FUNCTION Filtro : REAL
VAR_INPUT
	Input:REAL;	//Entrada do sensor
	Tempo:DINT := 500;	//Tempo de amostragem
END_VAR
VAR
	Amostras:ARRAY[1..50] OF REAL;
	TON_Amostras:TON;
	i		:INT;	//Variável de iteração do FOR
	Soma 	:REAL;	//Somatório dos valores do array
	Teste: INT;
END_VAR

TON_Amostras(IN := NOT TON_Amostras.Q, PT:=DINT_TO_TIME(Tempo));

IF TON_Amostras.Q THEN
	//Faz o shift do array
	FOR i := 1 TO 49 DO
		Amostras[i] := Amostras[i + 1];
	END_FOR
	
	//Insere a leitura do sensor na última posição
	Amostras[50] := Input;
	
	//Soma os valores do array
	Soma := 0;
	FOR i := 1 TO 50 DO
		Soma := Soma + Amostras[i];
	END_FOR
	
	Filtro := Soma / 50;
	
END_IF

END_FUNCTION

(* stored: Version 1.1.0.1, ProductVersion 3.1.4024.14
   POU Filtro: Id {06e7fbb2-e038-45fb-a9df-a42eac37f878}, SpecialFunc None *)
